PROGRAM Manual
VAR
	running: BOOL;
	currentError: UDINT;
	manualMode: E_JogMode;
	velocity: LREAL;
	acceleration: LREAL;
	deceleration: LREAL;
	jerk: LREAL;
	done: BOOL;
	busy: BOOL;
	reset: BOOL;
END_VAR

HAVL.axis.ReadStatus();


HAVL.axisPower(
	Axis:= HAVL.axis,
	Enable:= HAVL.enable,
	Enable_Positive:= HAVL.enable,
	Enable_Negative:= HAVL.enable,
	Override:= HAVL.override,
	BufferMode:= ,
	Options:= ,
	Status=> HAVL.running,
	Busy=> ,
	Active=> ,
	Error=> ,
	ErrorID=> currentError
);

HAVL.axisMoveManual(
	Axis:= HAVL.axis,
	JogForward:= HAVL.forward,
	JogBackwards:= HAVL.backwards,
	Mode:= ,
	Position:= ,
	Velocity:= ,
	Acceleration:= ,
	Deceleration:= ,
	Jerk:= ,
	Done=> HAVL.done,
	Busy=> HAVL.busy,
	Active=> ,
	CommandAborted=> ,
	Error=> ,
	ErrorID=> );
	
IF HAVL.busy THEN
	HAVL.axisReadActualPosition(Axis := HAVL.axis, Enable := TRUE, Valid=>, Busy=>, Error=>, ErrorID=>, Position=> HAVL.actualPosition);
END_IF
HAVL.actualPositionInt := LREAL_TO_INT(HAVL.actualPosition);

HAVL.axisErrorReset(Axis := HAVL.axis, Execute := HAVL.resetError, Done =>, Error =>, ErrorID => currentError);

END_PROGRAM

(* stored: Version 1.1.0.1, ProductVersion 3.1.4024.6
   POU Manual: Id {880819fa-648e-4916-b2f4-018c51c85792}, SpecialFunc None *)
